{attribute 'global_init_slot' := '49991'}
{attribute 'qualified_only'}
VAR_GLOBAL
	// encoder resolution
	g_incEncoderRes :ARRAY[1..g_sArmNum,1..g_sJntNum] OF DINT;
	g_absEncoderRes :ARRAY[1..g_sArmNum,1..g_sJntNum] OF DINT;
	
	// reduction ratio
	g_motorReduction :ARRAY[1..g_sArmNum,1..g_sJntNum] OF LREAL;
	g_absEncoderReduction :ARRAY[1..g_sArmNum,1..g_sJntNum] OF LREAL;
	
	// motor parameters
	g_motorTrqConst :ARRAY[1..g_sArmNum,1..g_sJntNum] OF LREAL;
	g_motorMaxCurrent :ARRAY[1..g_sArmNum,1..g_sJntNum] OF LREAL;//mA
	
	// motor encoder direction
	g_motorDir :ARRAY[1..g_sJntNum] OF INT ;
																 
	// joint position limit
	g_minJntPos: ARRAY[1..g_sJntNum] OF LREAL;	
	g_maxJntPos: ARRAY[1..g_sJntNum] OF LREAL;
	
	// DH joint position limit
	//NOTE: wrist pitch and yaw angle is reset after instrument is mounted 
	g_minDHJntPos : ARRAY[1..6] OF LREAL;
	g_maxDHJntPos : ARRAY[1..6] OF LREAL;
	
	// joint velocity limit
	g_maxJntVel :ARRAY[1..g_sJntNum] OF LREAL;

	// joint position at link encoder calibrated point
	g_linkEncCaliJntPos :ARRAY[1..g_sJntNum] OF LREAL;
	
	// absolute encoder direction
	g_asbEncoderDir :ARRAY[1..g_sJntNum] OF INT;
		
	// minimum distance between instrument/endoscope tip and remote center
	g_minInstruRCDis:LREAL;
	g_minScopeRCDis:LREAL;	
	
END_VAR

(* stored: Version 1.1.0.1, ProductVersion 3.1.4024.11
   GVL GVL_SlaveMotorParameters: Id {cf487053-15bb-46bd-a4ed-bbb1df690beb} *)
